// TIA Portal V21 export
DATA_BLOCK "Additivo"   // DB13
{ S7_Optimized_Access := 'TRUE' }
// stored: MemoryReserve 100
   VAR
      "A" : Array[0.."K_NumAdditivo"] of "Std_Additivo";
   END_VAR
BEGIN
   "A"[0].Attuale := 0.0;
   "A"[0].Allarme := FALSE;
END_DATA_BLOCK
